// TIA Portal V20 export
DATA_BLOCK "IDB_LineC1"   // DB10
// stored: InstanceOfName LineC1.FB_LineC1, InstanceOfType FB, Namespace LineC1
"LineC1.FB_LineC1"
   // VAR
   //    "Conveyor_C1.1.1" : "Global.FB_Conveyor";
   //    "Conveyor_C1.1.2" { S7_SetPoint := 'True'} : "Global.FB_Conveyor";
   //    "Conveyor_C1.1.3" { S7_SetPoint := 'True'} : "Global.FB_Conveyor";
   //    "MABS_C1.2.1" : "Global.FB_MABS";
   //    "MABS_C1.2.2" { S7_SetPoint := 'True'} : "Global.FB_MABS";
   //    "Conveyor_C1.3.1" { S7_SetPoint := 'True'} : "Global.FB_Conveyor";
   //    "Conveyor_C1.3.2" { S7_SetPoint := 'True'} : "Global.FB_Conveyor";
   //    "Conveyor_C1.3.3" { S7_SetPoint := 'True'} : "Global.FB_Conveyor";
   //    "Conveyor_C1.3.4" { S7_SetPoint := 'True'} : "Global.FB_Conveyor";
   //    "Conveyor_C1.3.5" { S7_SetPoint := 'True'} : "Global.FB_Conveyor";
   //    "Conveyor_C1.3.6" { S7_SetPoint := 'True'} : "Global.FB_Conveyor";
   //    "Conveyor_C1.3.7" { S7_SetPoint := 'True'} : "Global.FB_Conveyor";
   //    "Conveyor_C1.3.8" { S7_SetPoint := 'True'} : "Global.FB_Conveyor";
   //    "Conveyor_C1.3.9" { S7_SetPoint := 'True'} : "Global.FB_Conveyor";
   //    "Conveyor_C1.3.10" { S7_SetPoint := 'True'} : "Global.FB_Conveyor";
   //    "Conveyor_C1.4.1" { S7_SetPoint := 'True'} : "Global.FB_Conveyor";
   //    "Conveyor_C1.4.2" { S7_SetPoint := 'True'} : "Global.FB_Conveyor";
   //    "Conveyor_C1.4.3" { S7_SetPoint := 'True'} : "Global.FB_Conveyor";
   //    "Conveyor_C1.4.4" { S7_SetPoint := 'True'} : "Global.FB_Conveyor";
   //    "Conveyor_C1.5.1" { S7_SetPoint := 'True'} : "Global.FB_Conveyor";
   //    "Conveyor_C1.6.1" { S7_SetPoint := 'True'} : "Global.FB_Conveyor";
   //    "Conveyor_C1.6.2" { S7_SetPoint := 'True'} : "Global.FB_Conveyor";
   //    "Conveyor_C1.7.1" { S7_SetPoint := 'True'} : "Global.FB_Conveyor";
   //    "Conveyor_C1.7.2" { S7_SetPoint := 'True'} : "Global.FB_Conveyor";
   //    "Conveyor_C1.7.3" { S7_SetPoint := 'True'} : "Global.FB_Conveyor";
   //    "Conveyor_C1.7.4" { S7_SetPoint := 'True'} : "Global.FB_Conveyor";
   //    "Conveyor_C1.7.5" { S7_SetPoint := 'True'} : "Global.FB_Conveyor";
   //    "Conveyor_C1.7.6" { S7_SetPoint := 'True'} : "Global.FB_Conveyor";
   //    "Conveyor_C1.7.7" { S7_SetPoint := 'True'} : "Global.FB_Conveyor";
   //    "Conveyor_C1.7.8" { S7_SetPoint := 'True'} : "Global.FB_Conveyor";
   //    "Conveyor_C1.7.9" { S7_SetPoint := 'True'} : "Global.FB_Conveyor";
   //    "Conveyor_C1.7.10" { S7_SetPoint := 'True'} : "Global.FB_Conveyor";
   //    "Conveyor_C1.8.0" { S7_SetPoint := 'True'} : "Global.FB_Conveyor";
   //    "Conveyor_C1.9.1" { S7_SetPoint := 'True'} : "Global.FB_Conveyor";
   //    "Conveyor_C1.10.1" { S7_SetPoint := 'True'} : "Global.FB_Conveyor";
   //    "Conveyor_C1.11.1" { S7_SetPoint := 'True'} : "Global.FB_Conveyor";
   //    "Conveyor_C1.11.2" { S7_SetPoint := 'True'} : "Global.FB_Conveyor";
   //    "Conveyor_C1.12.1" { S7_SetPoint := 'True'} : "Global.FB_Conveyor";
   //    "Conveyor_C1.12.2" { S7_SetPoint := 'True'} : "Global.FB_Conveyor";
   //    "Conveyor_C1.12.3" { S7_SetPoint := 'True'} : "Global.FB_Conveyor";
   //    "Transfer_C1.13.1" : "Global.FB_S300_tTransMode";
   //    "Transfer_C1.14.1" { S7_SetPoint := 'True'} : "Global.FB_S300_tTransMode";
   //    "Conveyor_C1.15.2" { S7_SetPoint := 'True'} : "Global.FB_Conveyor";
   //    "Conveyor_C1.15.3" { S7_SetPoint := 'True'} : "Global.FB_Conveyor";
   //    "Conveyor_C1.15.4" { S7_SetPoint := 'True'} : "Global.FB_Conveyor";
   //    "Conveyor_C1.16.1" { S7_SetPoint := 'True'} : "Global.FB_Conveyor";
   //    "Conveyor_C1.17.0" { S7_SetPoint := 'True'} : "Global.FB_Conveyor";
   //    "Conveyor_C1.18.1" { S7_SetPoint := 'True'} : "Global.FB_Conveyor";
   //    "Conveyor_C1.18.2" { S7_SetPoint := 'True'} : "Global.FB_Conveyor";
   //    "Conveyor_C1.18.3" { S7_SetPoint := 'True'} : "Global.FB_Conveyor";
   //    "Conveyor_C1.18.4" { S7_SetPoint := 'True'} : "Global.FB_Conveyor";
   //    "Conveyor_C1.18.5" { S7_SetPoint := 'True'} : "Global.FB_Conveyor";
   //    "Conveyor_C1.18.6" { S7_SetPoint := 'True'} : "Global.FB_Conveyor";
   //    "Conveyor_C1.18.7" { S7_SetPoint := 'True'} : "Global.FB_Conveyor";
   //    "Conveyor_C1.19.1" { S7_SetPoint := 'True'} : "Global.FB_Conveyor";
   //    "Conveyor_C1.20.2" { S7_SetPoint := 'True'} : "Global.FB_Conveyor";
   // END_VAR
BEGIN
END_DATA_BLOCK
